METHOD INTERNAL ParseResponsePayload : DINT
VAR_INPUT
  /// Response data
  ResponseData : RobotLibraryRecvDataFB;
  /// Timestamp
  Timestamp    : SystemTime;  
END_VAR
// Table 6-147: Received CMD payload (RC to PLC) of "WriteRobotDefaultDynamics"
// --------------------------
// Header
// --------------------------
// Byte 00 : USINT   - ParSeq | State     
// Byte 01 : SINT    - AlarmMessageSeverity    
// Byte 02 : UINT    - AlarmMessageCode HB
// Byte 03 :         - AlarmMessageCode LB
// --------------------------
// Datablock
// --------------------------
// Byte 04 : UINT VelocityRate
// Byte 05 : 
// Byte 06 : UINT AccelerationRate
// Byte 07 : 
// Byte 08 : UINT DecelerationRate
// Byte 09 : 
// Byte 10 : UINT JerkRate
// Byte 11 : 
// --------------------------
// call base implementation to parse the header from payload buffer
ResponseData.PayloadPtr := SUPER^.ParseResponsePayload(ResponseData := ResponseData, Timestamp := Timestamp);

// copy parsed header to response
_response.ParSeq               := _rspHeader.ParSeq;
_response.State                := _rspHeader.State;
_response.AlarmMessageSeverity := _rspHeader.AlarmMessageSeverity;
_response.AlarmMessageCode     := _rspHeader.AlarmMessageCode;

// Get Response.VelocityRate
_response.VelocityRate     := ResponseData.GetUint();
// Get Response.AccelerationRate
_response.AccelerationRate := ResponseData.GetUint();
// Get Response.DecelerationRate
_response.DecelerationRate := ResponseData.GetUint();
// Get Response.JerkRate
_response.JerkRate         := ResponseData.GetUint();

// Create logging
ParseResponsePayloadLog(ResponseData := ResponseData, Timestamp := Timestamp);
END_METHOD

METHOD INTERNAL ParseResponsePayloadLog
VAR_INPUT
  /// Response data
  ResponseData : RobotLibraryRecvDataFB;
  /// Timestamp
  Timestamp    : SystemTime;  
END_VAR
// Create log entry for Parameter start
CreateLogMessage      ( Timestamp   := Timestamp,
                        MessageType := MessageType.CMD,
                        Severity    := Severity.DEBUG,
                        MessageCode := 0,
                        MessageText := 'Parsed the following parameter(s) from response data:');
               
// Create log entry for VelocityRate
CreateLogMessagePara1 ( Timestamp   := Timestamp,
                        MessageType := MessageType.CMD,
                        Severity    := Severity.DEBUG,
                        MessageCode := 0,
                        MessageText := 'Response.VelocityRate = {1}',
                        Para1       :=  UINT_TO_STRING(_response.VelocityRate));

// Create log entry for AccelerationRate
CreateLogMessagePara1 ( Timestamp   := Timestamp,
                        MessageType := MessageType.CMD,
                        Severity    := Severity.DEBUG,
                        MessageCode := 0,
                        MessageText := 'Response.AccelerationRate = {1}',
                        Para1       :=  UINT_TO_STRING(_response.AccelerationRate));

// Create log entry for DecelerationRate
CreateLogMessagePara1 ( Timestamp   := Timestamp,
                        MessageType := MessageType.CMD,
                        Severity    := Severity.DEBUG,
                        MessageCode := 0,
                        MessageText := 'Response.DecelerationRate = {1}',
                        Para1       :=  UINT_TO_STRING(_response.DecelerationRate));

// Create log entry for JerkRate
CreateLogMessagePara1 ( Timestamp   := Timestamp,
                        MessageType := MessageType.CMD,
                        Severity    := Severity.DEBUG,
                        MessageCode := 0,
                        MessageText := 'Response.JerkRate = {1}',
                        Para1       :=  UINT_TO_STRING(_response.JerkRate));
END_METHOD

METHOD PROTECTED Reset : DINT
VAR_INPUT
END_VAR
Reset := SUPER^.Reset();

Done               := FALSE;
Busy               := FALSE;
CommandBuffered    := FALSE;
CommandAborted     := FALSE;
CommandInterrupted := FALSE;
END_METHOD

END_FUNCTION_BLOCK

// Library/POUs/Write/MC_WriteRobotReferenceDynamics/MC_WriteRobotReferenceDynamicsFB
/// Write reference values of robot dynamics for path movement
FUNCTION_BLOCK MC_WriteRobotReferenceDynamicsFB EXTENDS RobotLibraryBaseExecuteFB
// ------------------------------------------------------------------------- 
//  SRCI Robot Library                                                
// ------------------------------------------------------------------------- 
//                                                                           
//  Object:      WriteRobotReferenceDynamicsFB                                       
//  Author:      Thorsten Brach                                                
//  Date:        2024-06-01
//
//  Description:                                              
//   
//                                                                           
//  Copyright: 
//    (C) 2024 Thorsten Brach. All rights reserved                                                                                                                                            
//             Licensed under the LGPL-3.0 license.
//                                                                           
//  Disclaimer:                                                                           
//    This project is provided without any guarantee and can be used for   
//    private and commercial purposes. Any use is at the user’s 
//    own risk and responsibility.
//
// -------------------------------------------------------------------------
VAR_INPUT
  /// Processing Mode
  ProcessingMode     : ProcessingMode;
  /// internal copy of command parameter 
  ParCmd             : WriteRobotReferenceDynamicsParCmd; 
END_VAR
VAR_OUTPUT
  /// Command is transferred and confirmed by the RC
  CommandBuffered    : BOOL;
  /// The command was aborted by another command
  CommandAborted     : BOOL;
  /// TRUE, while command is interrupted during execution and can be continued.
  CommandInterrupted : BOOL;
  /// command outputs
  OutCmd             : WriteRobotReferenceDynamicsOutCmd;       
END_VAR

VAR
  /// internal copy of command parameter 
 _parCmd             : WriteRobotReferenceDynamicsParCmd;
  /// command data to send
 _command            : WriteRobotReferenceDynamicsSendData;
  /// response data received
 _response           : WriteRobotReferenceDynamicsRecvData;      
END_VAR

SUPER^(AxesGroup := AxesGroup);

METHOD PROTECTED CheckFunctionSupported : BOOL
VAR_IN_OUT
  /// Robot assignment of function
  AxesGroup : AxesGroup; 
END_VAR
CheckFunctionSupported := AxesGroup.InternalData.RCSupportedFunctions.WriteRobotReferenceDynamics;

IF ( NOT CheckFunctionSupported )
THEN
  // call base implementation for set error and create log entry
  SUPER^.CheckFunctionSupported(AxesGroup := AxesGroup);
END_IF
END_METHOD

METHOD PROTECTED CheckParameterChanged : BOOL
VAR_IN_OUT
  /// Robot assignment of function
  AxesGroup    : AxesGroup; 
END_VAR
// Check ParCmd Size is > 0, because MemCmp does not work correctly with size = 0
IF (SIZEOF(ParCmd) = 0) 
THEN 
  RETURN;
END_IF

// compare memory 
_parameterChanged := ( SysDepMemCmp(pData1 := ADR(ParCmd), pData2 := ADR(_parCmd), DataLen := SIZEOF(ParCmd)) <> RobotLibraryConstants.OK );

// check parameter valid ?
_parameterValid   := CheckParameterValid( AxesGroup := AxesGroup );

IF ((  _parameterChanged        )  AND 
    (  _parameterValid          )) OR
    (  _parameterUpdateInternal )  
THEN  
  // reset internal flag for send parameter update
 _parameterUpdateInternal := FALSE;
  // update internal copy of parameters 
 _parCmd := ParCmd;
  // inc parameter sequence
 _command.ParSeq := _command.ParSeq + 1;
  // update command data  
  CommandData := CreateCommandPayload(AxesGroup := AxesGroup); // ( Access via reference to rCommandFB in ACR )
  // notify active command register 
  AxesGroup.Acyclic.ActiveCommandRegister.NotifyParameterChanged := _uniqueID;
END_IF
END_METHOD

METHOD INTERNAL CreateCommandPayload : RobotLibrarySendDataFB
VAR_IN_OUT
  /// Robot assignment of function
  AxesGroup : AxesGroup; 
END_VAR
// Table 6-139: Sent CMD payload (PLC to RC) of "WriteRobotReferenceDynamics"
// --------------------------
// Header
// --------------------------
// Byte 00 : UINT  - Type HB     
// Byte 01 :       - Type LB    
// Byte 02 : USINT - Reserve | ExecutionMode
// Byte 03 : USINT - ParSeq  | Priority
// --------------------------
// Datablock
// --------------------------
// Byte 04 : DATE Date
// Byte 05 : 
// Byte 06 : TIME_OF_DAY Time
// Byte 07 : 
// Byte 08 : 
// Byte 09 : REAL VelocityReference
// Byte 10 : 
// Byte 11 : 
// Byte 12 : REAL AccelerationReference
// Byte 13 : 
// Byte 14 : 
// Byte 15 : REAL DecelerationReference
// Byte 16 : 
// Byte 17 : 
// Byte 18 : REAL JerkReference
// Byte 19 : 
// Byte 20 : 
// Byte 21 : 
// Byte 22 : REAL 
// Byte 23 : 
// Byte 24 : 
// Byte 25 : 
// --------------------------
// set command parameter 
_command.CmdTyp                :=  CmdType.WriteRobotReferenceDynamics;
_command.ExecMode              :=  ExecMode;
_command.ParSeq                := _command.ParSeq;
_command.Priority              :=  Priority;

_command.DynamicValues         := _parCmd.DynamicValues; {warning 'ToDo: Check if this is a mistake in the SRCI specification ? '}

(*
 _command.Timestamp             := _parCmd.DynamicValues.Timestamp;
 _command.VelocityReference     := REAL_TO_PERCENT_UINT(_parCmd.DynamicValues.VelocityReference     , IsOptional := FALSE);
 _command.AccelerationReference := REAL_TO_PERCENT_UINT(_parCmd.DynamicValues.AccelerationReference , IsOptional := FALSE);
 _command.JerkReference         := REAL_TO_PERCENT_UINT(_parCmd.DynamicValues.JerkReference         , IsOptional := TRUE );
 _command.DecelerationReference := REAL_TO_PERCENT_UINT(_parCmd.DynamicValues.DecelerationReference , IsOptional := TRUE );
*)


// copy command data to header
_cmdHeader := _command;
// call base implementation to copy header to payload buffer
CreateCommandPayload := SUPER^.CreateCommandPayload(AxesGroup := AxesGroup);

// add command.DynamicValues.Timestamp.IEC_DATE
CreateCommandPayload.AddUint(_command.DynamicValues.Timestamp.IEC_DATE);
// add command.DynamicValues.Timestamp.IEC_TIME
CreateCommandPayload.AddTime(_command.DynamicValues.Timestamp.IEC_TIME);
// add command.DynamicValues.VelocityReference
CreateCommandPayload.AddReal(_command.DynamicValues.VelocityReference);
// add command.DynamicValues.AccelerationReference
CreateCommandPayload.AddReal(_command.DynamicValues.AccelerationReference);
// add command.DynamicValues.DecelerationRate
CreateCommandPayload.AddReal(_command.DynamicValues.DecelerationReference);
// add command.DynamicValues.JerkRate
CreateCommandPayload.AddReal(_command.DynamicValues.JerkReference);

// Create logging
CreateCommandPayloadLog(AxesGroup := AxesGroup);
END_METHOD

METHOD INTERNAL CreateCommandPayloadLog
VAR_IN_OUT
  /// Robot assignment of function
  AxesGroup : AxesGroup; 
END_VAR
// Create log entry for Parameter start
CreateLogMessage      ( Timestamp   := AxesGroup.InternalData.SystemTime,
                        MessageType := MessageType.CMD,
                        Severity    := Severity.DEBUG,
                        MessageCode := 0,
                        MessageText := 'Create command payload with the following parameter(s) :');
  
// Create log entry for DynamicValues.Timestamp.IEC_DATE
CreateLogMessagePara1 ( Timestamp   := AxesGroup.InternalData.SystemTime,
                        MessageType := MessageType.CMD,
                        Severity    := Severity.DEBUG,
                        MessageCode := 0,
                        MessageText := 'Command.DynamicValues.Timestamp.IEC_DATE = {1}',
                        Para1       :=  IEC_DATE_TO_STRING(_command.DynamicValues.Timestamp.IEC_DATE));

// Create log entry for DynamicValues.Timestamp.IEC_TIME
CreateLogMessagePara1 ( Timestamp   := AxesGroup.InternalData.SystemTime,
                        MessageType := MessageType.CMD,
                        Severity    := Severity.DEBUG,
                        MessageCode := 0,
                        MessageText := 'Command.DynamicValues.Timestamp.IEC_TIME = {1}',
                        Para1       :=  IEC_TIME_TO_STRING(_command.DynamicValues.Timestamp.IEC_TIME));

// Create log entry for DynamicValues.VelocityReference
CreateLogMessagePara1 ( Timestamp   := AxesGroup.InternalData.SystemTime,
                        MessageType := MessageType.CMD,
                        Severity    := Severity.DEBUG,
                        MessageCode := 0,
                        MessageText := 'Command..DynamicValues.VelocityReference = {1}',
                        Para1       :=  REAL_TO_STRING(_command.DynamicValues.VelocityReference));

// Create log entry for DynamicValues.AccelerationReference
CreateLogMessagePara1 ( Timestamp   := AxesGroup.InternalData.SystemTime,
                        MessageType := MessageType.CMD,
                        Severity    := Severity.DEBUG,
                        MessageCode := 0,
                        MessageText := 'Command.DynamicValues.AccelerationReference = {1}',
                        Para1       :=  REAL_TO_STRING(_command.DynamicValues.AccelerationReference));

// Create log entry for DynamicValues.DecelerationReference
CreateLogMessagePara1 ( Timestamp   := AxesGroup.InternalData.SystemTime,
                        MessageType := MessageType.CMD,
                        Severity    := Severity.DEBUG,
                        MessageCode := 0,
                        MessageText := 'Command.DynamicValues.DecelerationReference = {1}',
                        Para1       :=  REAL_TO_STRING(_command.DynamicValues.DecelerationReference));

// Create log entry for DynamicValues.JerkReference
CreateLogMessagePara1 ( Timestamp   := AxesGroup.InternalData.SystemTime,
                        MessageType := MessageType.CMD,
                        Severity    := Severity.DEBUG,
                        MessageCode := 0,
                        MessageText := 'Command.DynamicValues.JerkReference = {1}',
                        Para1       :=  REAL_TO_STRING(_command.DynamicValues.JerkReference));
END_METHOD

METHOD FB_init : BOOL
VAR_INPUT
  /// if TRUE, the retain variables are initialized (warm start / cold start)
  bInitRetains : BOOL; 
  /// if TRUE, the instance afterwards gets moved into the copy code (online change)
  bInCopyCode  : BOOL;  
END_VAR
MyType := 'MC_WriteRobotReferenceDynamicsFB';

ExecMode := ExecutionMode.PARALLEL;
END_METHOD

METHOD PROTECTED OnCall
VAR_IN_OUT
  /// Robot assignment of function
  AxesGroup : AxesGroup; 
END_VAR
// call base implementation
SUPER^.OnCall(AxesGroup := AxesGroup);

CASE _stepCmd OF
  
  00:  IF ( _execute_R.Q )  
       THEN
         // Check function is supported and parameter are valid ?
         IF (( CheckFunctionSupported( AxesGroup := AxesGroup )) AND
             ( CheckParameterValid   ( AxesGroup := AxesGroup )))
         THEN      
           // set busy flag
           Busy := TRUE;
           // Reset command outputs
           SysDepMemSet(pDest := ADR(OutCmd), Value := 0, DataLen := SIZEOF(OutCmd));         
           // apply command parameter
          _parCmd := ParCmd;
           // init parameter sequence
          _command.ParSeq := 1;
           // create command data
           CommandData := CreateCommandPayload(AxesGroup := AxesGroup);
           // Add command to active command register
          _uniqueID := AxesGroup.Acyclic.ActiveCommandRegister.AddCmd( pCommandFB := ADR(THIS^ ));     
           // set timeout
           SetTimeout(PT := _timeoutCmd, rTimer := _timerCmd);
           // inc step counter
          _stepCmd := _stepCmd + 1;
         END_IF 
       END_IF
     

  01:  // Wait for responce received
       IF ( _responseReceived )
       THEN
         // reset response received flag
        _responseReceived := FALSE;

         CASE  _response.State 
         OF
           CmdMessageState.BUFFERED    : CommandBuffered    := TRUE;
           CmdMessageState.INTERRUPTED : CommandInterrupted := TRUE;           
           CmdMessageState.DONE        : Done               := TRUE;           
           CmdMessageState.ABORTED     : CommandAborted     := TRUE;
           CmdMessageState.ERROR       : Error              := TRUE;
         END_CASE
                
         // Done, Aborted or Error ?
         IF (_response.State >= CmdMessageState.DONE )
         THEN
           // Reset Busy flag
           Busy := FALSE;
           // Update results
           OutCmd.ReferenceDynamicValues.VelocityReference     := _response.ReferenceDynamicValues.VelocityReference; 
           OutCmd.ReferenceDynamicValues.AccelerationReference := _response.ReferenceDynamicValues.AccelerationReference;
           OutCmd.ReferenceDynamicValues.DecelerationReference := _response.ReferenceDynamicValues.DecelerationReference;
           OutCmd.ReferenceDynamicValues.JerkReference         := _response.ReferenceDynamicValues.JerkReference;

           // set timeout
           SetTimeout(PT := _timeoutCmd, rTimer := _timerCmd);
           // inc step counter
          _stepCmd := _stepCmd + 1; 
         END_IF
       END_IF


  02: IF ( NOT Execute)
      THEN
        Reset();
      END_IF     

ELSE
  // invalid step
  ErrorID := RobotLibraryEvents.ERR_INVALID_STEP;
END_CASE


// Reset FB
IF ( NOT Execute )
THEN
  Reset();
END_IF
END_METHOD

METHOD INTERNAL ParseResponsePayload : DINT
VAR_INPUT
  /// Response data
  ResponseData : RobotLibraryRecvDataFB;
  /// Timestamp
  Timestamp    : SystemTime;  
END_VAR
// Table 6-140: Received CMD payload (RC to PLC) of "WriteRobotReferenceDynamics"
// --------------------------
// Header
// --------------------------
// Byte 00 : USINT   - ParSeq | State     
// Byte 01 : SINT    - AlarmMessageSeverity    
// Byte 02 : UINT    - AlarmMessageCode HB
// Byte 03 :         - AlarmMessageCode LB
// --------------------------
// Datablock
// --------------------------
// Byte 04 : REAL VelocityReference
// Byte 05 : 
// Byte 06 : 
// Byte 07 : 
// Byte 08 : REAL AccelerationReference
// Byte 09 : 
// Byte 10 : 
// Byte 11 : 
// Byte 12 : REAL DecelerationReference
// Byte 13 : 
// Byte 14 : 
// Byte 15 : 
// Byte 16 : REAL JerkReference
// Byte 17 : 
// Byte 18 : 
// Byte 19 : 
// --------------------------
// call base implementation to parse the header from payload buffer
ResponseData.PayloadPtr := SUPER^.ParseResponsePayload(ResponseData := ResponseData, Timestamp := Timestamp);

// copy parsed header to response
_response.ParSeq               := _rspHeader.ParSeq;
_response.State                := _rspHeader.State;
_response.AlarmMessageSeverity := _rspHeader.AlarmMessageSeverity;
_response.AlarmMessageCode     := _rspHeader.AlarmMessageCode;

// Get Response.ReferenceDynamicValues.VelocityReference
_response.ReferenceDynamicValues.VelocityReference := ResponseData.GetReal();
// Get Response.ReferenceDynamicValues.AccelerationReference
_response.ReferenceDynamicValues.AccelerationReference := ResponseData.GetReal();
// Get Response.ReferenceDynamicValues.DecelerationReference
_response.ReferenceDynamicValues.DecelerationReference := ResponseData.GetReal();
// Get ReferenceDynamicValues.JerkReference
_response.ReferenceDynamicValues.JerkReference := ResponseData.GetReal();

// Create logging
ParseResponsePayloadLog(ResponseData := ResponseData, Timestamp := Timestamp);
END_METHOD

METHOD INTERNAL ParseResponsePayloadLog
VAR_INPUT
  /// Response data
  ResponseData : RobotLibraryRecvDataFB;
  /// Timestamp
  Timestamp    : SystemTime;  
END_VAR
// Create log entry for Parameter start
CreateLogMessage      ( Timestamp   := Timestamp,
                        MessageType := MessageType.CMD,
                        Severity    := Severity.DEBUG,
                        MessageCode := 0,
                        MessageText := 'Parsed the following parameter(s) from response data:');

// Create log entry for ReferenceDynamicValues.VelocityReference
CreateLogMessagePara1 ( Timestamp   := Timestamp,
                        MessageType := MessageType.CMD,
                        Severity    := Severity.DEBUG,
                        MessageCode := 0,
                        MessageText := 'Response.ReferenceDynamicValues.VelocityReference = {1}',
                        Para1       :=  REAL_TO_STRING(_response.ReferenceDynamicValues.VelocityReference));

// Create log entry for ReferenceDynamicValues.AccelerationReference
CreateLogMessagePara1 ( Timestamp   := Timestamp,
                        MessageType := MessageType.CMD,
                        Severity    := Severity.DEBUG,
                        MessageCode := 0,
                        MessageText := 'Response.ReferenceDynamicValues.AccelerationReference = {1}',
                        Para1       :=  REAL_TO_STRING(_response.ReferenceDynamicValues.AccelerationReference));
                        
// Create log entry for ReferenceDynamicValues.DecelerationReference
CreateLogMessagePara1 ( Timestamp   := Timestamp,
                        MessageType := MessageType.CMD,
                        Severity    := Severity.DEBUG,
                        MessageCode := 0,
                        MessageText := 'Response.ReferenceDynamicValues.DecelerationReference = {1}',
                        Para1       :=  REAL_TO_STRING(_response.ReferenceDynamicValues.DecelerationReference));

// Create log entry for ReferenceDynamicValues.JerkReference
CreateLogMessagePara1 ( Timestamp   := Timestamp,
                        MessageType := MessageType.CMD,
                        Severity    := Severity.DEBUG,
                        MessageCode := 0,
                        MessageText := 'Response.ReferenceDynamicValues.JerkReference = {1}',
                        Para1       :=  REAL_TO_STRING(_response.ReferenceDynamicValues.JerkReference));
END_METHOD

METHOD PROTECTED Reset : DINT
VAR_INPUT
END_VAR
Reset := SUPER^.Reset();

Done               := FALSE;
Busy               := FALSE;
CommandBuffered    := FALSE;
CommandAborted     := FALSE;
CommandInterrupted := FALSE;
END_METHOD

END_FUNCTION_BLOCK

// Library/POUs/Write/MC_WriteRobotSWLimits/MC_WriteRobotSWLimitsFB
/// Change robot limits of robot axes (degree)
FUNCTION_BLOCK MC_WriteRobotSWLimitsFB EXTENDS RobotLibraryBaseExecuteFB
// ------------------------------------------------------------------------- 
//  SRCI Robot Library                                                
// ------------------------------------------------------------------------- 
//                                                                           
//  Object:      WriteRobotSWLimitsFB                                       
//  Author:      Thorsten Brach                                                
//  Date:        2024-06-01
//
//  Description:                                              
//   
//                                                                           
//  Copyright: 
//    (C) 2024 Thorsten Brach. All rights reserved                                                                                                                                            
//             Licensed under the LGPL-3.0 license.
//                                                                           
//  Disclaimer:                                                                           
//    This project is provided without any guarantee and can be used for   
//    private and commercial purposes. Any use is at the user’s 
//    own risk and responsibility.
//
// -------------------------------------------------------------------------
VAR_INPUT
  /// command parameter 
  ParCmd          : WriteRobotSWLimitsParCmd;
END_VAR
VAR_OUTPUT
  /// Command is transferred and confirmed by the RC
  CommandBuffered : BOOL;
  /// command outputs
  OutCmd          : WriteRobotSWLimitsOutCmd;       
END_VAR

VAR
  /// internal copy of command parameter 
 _parCmd          : WriteRobotSWLimitsParCmd;
  /// command data to send
 _command         : WriteRobotSWLimitsSendData;
  /// response data received
 _response        : WriteRobotSWLimitsRecvData;      
END_VAR

SUPER^(AxesGroup := AxesGroup);

METHOD PROTECTED CheckFunctionSupported : BOOL
VAR_IN_OUT
  /// Robot assignment of function
  AxesGroup : AxesGroup; 
END_VAR
CheckFunctionSupported := AxesGroup.InternalData.RCSupportedFunctions.WriteRobotSWLimits;

IF ( NOT CheckFunctionSupported )
THEN
  // call base implementation for set error and create log entry
  SUPER^.CheckFunctionSupported(AxesGroup := AxesGroup);
END_IF
END_METHOD

METHOD PROTECTED CheckParameterChanged : BOOL
VAR_IN_OUT
  /// Robot assignment of function
  AxesGroup    : AxesGroup; 
END_VAR
// Check ParCmd Size is > 0, because MemCmp does not work correctly with size = 0
IF (SIZEOF(ParCmd) = 0) 
THEN 
  RETURN;
END_IF

// compare memory 
_parameterChanged := ( SysDepMemCmp(pData1 := ADR(ParCmd), pData2 := ADR(_parCmd), DataLen := SIZEOF(ParCmd)) <> RobotLibraryConstants.OK );

// check parameter valid ?
_parameterValid   := CheckParameterValid( AxesGroup := AxesGroup );

IF ((  _parameterChanged        )  AND 
    (  _parameterValid          )) OR
    (  _parameterUpdateInternal )  
THEN  
  // reset internal flag for send parameter update
 _parameterUpdateInternal := FALSE;
  // update internal copy of parameters 
 _parCmd := ParCmd;
  // inc parameter sequence
 _command.ParSeq := _command.ParSeq + 1;
  // update command data  
  CommandData := CreateCommandPayload(AxesGroup := AxesGroup); // ( Access via reference to rCommandFB in ACR )
  // notify active command register 
  AxesGroup.Acyclic.ActiveCommandRegister.NotifyParameterChanged := _uniqueID;
END_IF
END_METHOD

METHOD INTERNAL CreateCommandPayload : RobotLibrarySendDataFB
VAR_IN_OUT
  /// Robot assignment of function
  AxesGroup : AxesGroup; 
END_VAR
// Table 6-185: Sent CMD payload (PLC to RC) of "WriteRobotSWLimits"
// --------------------------
// Header
// --------------------------
// Byte 00 : UINT  - Type HB     
// Byte 01 :       - Type LB    
// Byte 02 : USINT - Reserve | ExecutionMode
// Byte 03 : USINT - ParSeq  | Priority
// --------------------------
// Datablock
// --------------------------
// Byte 04 : DATE Date
// Byte 05 : 
// Byte 06 : TIME_OF_DAY Time
// Byte 07 : 
// Byte 08 : 
// Byte 09 : REAL J1LowerLimit
// Byte 10 : 
// Byte 11 : 
// Byte 12 : REAL J2LowerLimit
// Byte 13 : 
// Byte 14 : 
// Byte 15 : REAL J3LowerLimit
// Byte 16 : 
// Byte 17 : 
// Byte 18 : REAL J4LowerLimit
// Byte 19 : 
// Byte 20 : 
// Byte 21 : REAL J5LowerLimit
// Byte 22 : 
// Byte 23 : 
// Byte 24 : REAL J6LowerLimit
// Byte 25 : 
// Byte 26 : 
// Byte 27 : REAL E1LowerLimit
// Byte 28 : 
// Byte 29 : 
// Byte 30 : REAL J1UpperLimit
// Byte 31 : 
// Byte 32 : 
// Byte 33 : REAL J2UpperLimit
// Byte 34 : 
// Byte 35 : 
// Byte 36 : REAL J3UpperLimit
// Byte 37 : 
// Byte 38 : 
// Byte 39 : REAL J4UpperLimit
// Byte 40 : 
// Byte 41 : 
// Byte 42 : REAL J5UpperLimit
// Byte 43 : 
// Byte 44 : 
// Byte 45 : REAL J6UpperLimit
// Byte 46 : 
// Byte 47 : 
// Byte 48 : REAL E1UpperLimit
// Byte 49 : 
// Byte 50 : 
// Byte 51 : REAL E2LowerLimit
// Byte 52 : 
// Byte 53 : 
// Byte 54 : REAL E3LowerLimit
// Byte 55 : 
// Byte 56 : 
// Byte 57 : REAL E4LowerLimit
// Byte 58 : 
// Byte 59 : 
// Byte 60 : REAL E5LowerLimit
// Byte 61 : 
// Byte 62 : 
// Byte 63 : REAL E6LowerLimit
// Byte 64 : 
// Byte 65 : 
// Byte 66 : REAL E2UpperLimit
// Byte 67 : 
// Byte 68 : 
// Byte 69 : REAL E3UpperLimit
// Byte 70 : 
// Byte 71 : 
// Byte 72 : REAL E4UpperLimit
// Byte 73 : 
// Byte 74 : 
// Byte 75 : REAL E5UpperLimit
// Byte 76 : 
// Byte 77 : 
// Byte 78 : REAL E6UpperLimit
// Byte 79 : 
// Byte 80 : 
// Byte 81 : 
// Byte 82 : BOOL ResetToFactoryDefault
// --------------------------
// set command parameter 
_command.CmdTyp                 :=  CmdType.WriteRobotSWLimits;
_command.ExecMode               :=  ExecMode;
_command.ParSeq                 := _command.ParSeq;
_command.Priority               :=  Priority;
                                
_command.LimitValues            :=  _parCmd.LimitValues;
_command.ResetToFactoryDefaults :=  _parCmd.ResetToFactoryDefaults;

// copy command data to header
_cmdHeader := _command;
// call base implementation to copy header to payload buffer
CreateCommandPayload := SUPER^.CreateCommandPayload(AxesGroup := AxesGroup);

// add command.LimitValues.Timestamp.IEC_DATE
CreateCommandPayload.AddUint(_command.LimitValues.Timestamp.IEC_DATE);
// add command.LimitValues.Timestamp.IEC_TIME
CreateCommandPayload.AddTime(_command.LimitValues.Timestamp.IEC_TIME);
// add command.LimitValues.J1LowerLimit
CreateCommandPayload.AddReal(_command.LimitValues.J1LowerLimit);
// add command.LimitValues.J2LowerLimit
CreateCommandPayload.AddReal(_command.LimitValues.J2LowerLimit);
// add command.LimitValues.J3LowerLimit
CreateCommandPayload.AddReal(_command.LimitValues.J3LowerLimit);
// add command.LimitValues.J41LowerLimit
CreateCommandPayload.AddReal(_command.LimitValues.J4LowerLimit);
// add command.LimitValues.J5LowerLimit
CreateCommandPayload.AddReal(_command.LimitValues.J5LowerLimit);
// add command.LimitValues.J6LowerLimit
CreateCommandPayload.AddReal(_command.LimitValues.J6LowerLimit);
// add command.LimitValues.E1LowerLimit
CreateCommandPayload.AddReal(_command.LimitValues.E1LowerLimit);
// add command.LimitValues.J1UpperLimit
CreateCommandPayload.AddReal(_command.LimitValues.J1UpperLimit);
// add command.LimitValues.J2UpperLimit
CreateCommandPayload.AddReal(_command.LimitValues.J2UpperLimit);
// add command.LimitValues.J3UpperLimit
CreateCommandPayload.AddReal(_command.LimitValues.J3UpperLimit);
// add command.LimitValues.J4UpperLimit
CreateCommandPayload.AddReal(_command.LimitValues.J4UpperLimit);
// add command.LimitValues.J5UpperLimit
CreateCommandPayload.AddReal(_command.LimitValues.J5UpperLimit);
// add command.LimitValues.J6UpperLimit
CreateCommandPayload.AddReal(_command.LimitValues.J6UpperLimit);
// add command.LimitValues.E1UpperLimit
CreateCommandPayload.AddReal(_command.LimitValues.E1UpperLimit);
// add command.LimitValues.E2LowerLimit
CreateCommandPayload.AddReal(_command.LimitValues.E2LowerLimit);
// add command.LimitValues.E3LowerLimit
CreateCommandPayload.AddReal(_command.LimitValues.E3LowerLimit);
// add command.LimitValues.E4LowerLimit
CreateCommandPayload.AddReal(_command.LimitValues.E4LowerLimit);
// add command.LimitValues.E5LowerLimit
CreateCommandPayload.AddReal(_command.LimitValues.E5LowerLimit);
// add command.LimitValues.E6LowerLimit
CreateCommandPayload.AddReal(_command.LimitValues.E6LowerLimit);
// add command.LimitValues.E2UpperLimit
CreateCommandPayload.AddReal(_command.LimitValues.E2UpperLimit);
// add command.LimitValues.E3UpperLimit
CreateCommandPayload.AddReal(_command.LimitValues.E3UpperLimit);
// add command.LimitValues.E4UpperLimit
CreateCommandPayload.AddReal(_command.LimitValues.E4UpperLimit);
// add command.LimitValues.E5UpperLimit
CreateCommandPayload.AddReal(_command.LimitValues.E5UpperLimit);
// add command.LimitValues.E6UpperLimit
CreateCommandPayload.AddReal(_command.LimitValues.E6UpperLimit);

// Create logging
CreateCommandPayloadLog(AxesGroup := AxesGroup);
END_METHOD

METHOD INTERNAL CreateCommandPayloadLog
VAR_IN_OUT
  /// Robot assignment of function
  AxesGroup : AxesGroup; 
END_VAR
// Create log entry for Parameter start
CreateLogMessage      ( Timestamp   := AxesGroup.InternalData.SystemTime,
                        MessageType := MessageType.CMD,
                        Severity    := Severity.DEBUG,
                        MessageCode := 0,
                        MessageText := 'Create command payload with the following parameter(s) :');
  
// Create log entry for LimitValues.Timestamp.IEC_DATE
CreateLogMessagePara1 ( Timestamp   := AxesGroup.InternalData.SystemTime,
                        MessageType := MessageType.CMD,
                        Severity    := Severity.DEBUG,
                        MessageCode := 0,
                        MessageText := 'Command.LimitValues.Timestamp.IEC_DATE = {1}',
                        Para1       :=  IEC_DATE_TO_STRING(_command.LimitValues.Timestamp.IEC_DATE));

// Create log entry for LimitValues.Timestamp.IEC_TIME
CreateLogMessagePara1 ( Timestamp   := AxesGroup.InternalData.SystemTime,
                        MessageType := MessageType.CMD,
                        Severity    := Severity.DEBUG,
                        MessageCode := 0,
                        MessageText := 'Command.LimitValues.Timestamp.IEC_TIME = {1}',
                        Para1       :=  IEC_TIME_TO_STRING(_command.LimitValues.Timestamp.IEC_TIME));

// Create log entry for LimitValues.J1LowerLimit
CreateLogMessagePara1 ( Timestamp   := AxesGroup.InternalData.SystemTime,
                        MessageType := MessageType.CMD,
                        Severity    := Severity.DEBUG,
                        MessageCode := 0,
                        MessageText := 'Command.LimitValues.J1LowerLimit = {1}',
                        Para1       :=  REAL_TO_STRING(_command.LimitValues.J1LowerLimit));

// Create log entry for LimitValues.J2LowerLimit
CreateLogMessagePara1 ( Timestamp   := AxesGroup.InternalData.SystemTime,
                        MessageType := MessageType.CMD,
                        Severity    := Severity.DEBUG,
                        MessageCode := 0,
                        MessageText := 'Command.LimitValues.J2LowerLimit = {1}',
                        Para1       :=  REAL_TO_STRING(_command.LimitValues.J2LowerLimit));
                        
// Create log entry for LimitValues.J3LowerLimit
CreateLogMessagePara1 ( Timestamp   := AxesGroup.InternalData.SystemTime,
                        MessageType := MessageType.CMD,
                        Severity    := Severity.DEBUG,
                        MessageCode := 0,
                        MessageText := 'Command.LimitValues.J3LowerLimit = {1}',
                        Para1       :=  REAL_TO_STRING(_command.LimitValues.J3LowerLimit));
                        
// Create log entry for LimitValues.J4LowerLimit
CreateLogMessagePara1 ( Timestamp   := AxesGroup.InternalData.SystemTime,
                        MessageType := MessageType.CMD,
                        Severity    := Severity.DEBUG,
                        MessageCode := 0,
                        MessageText := 'Command.LimitValues.J4LowerLimit = {1}',
                        Para1       :=  REAL_TO_STRING(_command.LimitValues.J4LowerLimit));

// Create log entry for LimitValues.J5LowerLimit
CreateLogMessagePara1 ( Timestamp   := AxesGroup.InternalData.SystemTime,
                        MessageType := MessageType.CMD,
                        Severity    := Severity.DEBUG,
                        MessageCode := 0,
                        MessageText := 'Command.LimitValues.J5LowerLimit = {1}',
                        Para1       :=  REAL_TO_STRING(_command.LimitValues.J5LowerLimit));

// Create log entry for LimitValues.J6LowerLimit
CreateLogMessagePara1 ( Timestamp   := AxesGroup.InternalData.SystemTime,
                        MessageType := MessageType.CMD,
                        Severity    := Severity.DEBUG,
                        MessageCode := 0,
                        MessageText := 'Command.LimitValues.J6LowerLimit = {1}',
                        Para1       :=  REAL_TO_STRING(_command.LimitValues.J6LowerLimit));

// Create log entry for LimitValues.E1LowerLimit
CreateLogMessagePara1 ( Timestamp   := AxesGroup.InternalData.SystemTime,
                        MessageType := MessageType.CMD,
                        Severity    := Severity.DEBUG,
                        MessageCode := 0,
                        MessageText := 'Command.LimitValues.E1LowerLimit = {1}',
                        Para1       :=  REAL_TO_STRING(_command.LimitValues.E1LowerLimit));

// Create log entry for LimitValues.J1UpperLimit
CreateLogMessagePara1 ( Timestamp   := AxesGroup.InternalData.SystemTime,
                        MessageType := MessageType.CMD,
                        Severity    := Severity.DEBUG,
                        MessageCode := 0,
                        MessageText := 'Command.LimitValues.J1UpperLimit = {1}',
                        Para1       :=  REAL_TO_STRING(_command.LimitValues.J1UpperLimit));

// Create log entry for LimitValues.J2UpperLimit
CreateLogMessagePara1 ( Timestamp   := AxesGroup.InternalData.SystemTime,
                        MessageType := MessageType.CMD,
                        Severity    := Severity.DEBUG,
                        MessageCode := 0,
                        MessageText := 'Command.LimitValues.J2UpperLimit = {1}',
                        Para1       :=  REAL_TO_STRING(_command.LimitValues.J2UpperLimit));

// Create log entry for LimitValues.J3UpperLimit
CreateLogMessagePara1 ( Timestamp   := AxesGroup.InternalData.SystemTime,
                        MessageType := MessageType.CMD,
                        Severity    := Severity.DEBUG,
                        MessageCode := 0,
                        MessageText := 'Command.LimitValues.J3UpperLimit = {1}',
                        Para1       :=  REAL_TO_STRING(_command.LimitValues.J3UpperLimit));

// Create log entry for LimitValues.J4UpperLimit
CreateLogMessagePara1 ( Timestamp   := AxesGroup.InternalData.SystemTime,
                        MessageType := MessageType.CMD,
                        Severity    := Severity.DEBUG,
                        MessageCode := 0,
                        MessageText := 'Command.LimitValues.J4UpperLimit = {1}',
                        Para1       :=  REAL_TO_STRING(_command.LimitValues.J4UpperLimit));

// Create log entry for LimitValues.J5UpperLimit
CreateLogMessagePara1 ( Timestamp   := AxesGroup.InternalData.SystemTime,
                        MessageType := MessageType.CMD,
                        Severity    := Severity.DEBUG,
                        MessageCode := 0,
                        MessageText := 'Command.LimitValues.J5UpperLimit = {1}',
                        Para1       :=  REAL_TO_STRING(_command.LimitValues.J5UpperLimit));

// Create log entry for LimitValues.J6UpperLimit
CreateLogMessagePara1 ( Timestamp   := AxesGroup.InternalData.SystemTime,
                        MessageType := MessageType.CMD,
                        Severity    := Severity.DEBUG,
                        MessageCode := 0,
                        MessageText := 'Command.LimitValues.J6UpperLimit = {1}',
                        Para1       :=  REAL_TO_STRING(_command.LimitValues.J6UpperLimit));

// Create log entry for LimitValues.E1UpperLimit
CreateLogMessagePara1 ( Timestamp   := AxesGroup.InternalData.SystemTime,
                        MessageType := MessageType.CMD,
                        Severity    := Severity.DEBUG,
                        MessageCode := 0,
                        MessageText := 'Command.LimitValues.E1UpperLimit = {1}',
                        Para1       :=  REAL_TO_STRING(_command.LimitValues.E1UpperLimit));

// Create log entry for LimitValues.E2LowerLimit
CreateLogMessagePara1 ( Timestamp   := AxesGroup.InternalData.SystemTime,
                        MessageType := MessageType.CMD,
                        Severity    := Severity.DEBUG,
                        MessageCode := 0,
                        MessageText := 'Command.LimitValues.E2LowerLimit = {1}',
                        Para1       :=  REAL_TO_STRING(_command.LimitValues.E2LowerLimit));

// Create log entry for LimitValues.E3LowerLimit
CreateLogMessagePara1 ( Timestamp   := AxesGroup.InternalData.SystemTime,
                        MessageType := MessageType.CMD,
                        Severity    := Severity.DEBUG,
                        MessageCode := 0,
                        MessageText := 'Command.LimitValues.E3LowerLimit = {1}',
                        Para1       :=  REAL_TO_STRING(_command.LimitValues.E3LowerLimit));

// Create log entry for LimitValues.E4LowerLimit
CreateLogMessagePara1 ( Timestamp   := AxesGroup.InternalData.SystemTime,
                        MessageType := MessageType.CMD,
                        Severity    := Severity.DEBUG,
                        MessageCode := 0,
                        MessageText := 'Command.LimitValues.E4LowerLimit = {1}',
                        Para1       :=  REAL_TO_STRING(_command.LimitValues.E4LowerLimit));

// Create log entry for LimitValues.E5LowerLimit
CreateLogMessagePara1 ( Timestamp   := AxesGroup.InternalData.SystemTime,
                        MessageType := MessageType.CMD,
                        Severity    := Severity.DEBUG,
                        MessageCode := 0,
                        MessageText := 'Command.LimitValues.E5LowerLimit = {1}',
                        Para1       :=  REAL_TO_STRING(_command.LimitValues.E5LowerLimit));

// Create log entry for LimitValues.E6LowerLimit
CreateLogMessagePara1 ( Timestamp   := AxesGroup.InternalData.SystemTime,
                        MessageType := MessageType.CMD,
                        Severity    := Severity.DEBUG,
                        MessageCode := 0,
                        MessageText := 'Command.LimitValues.E6LowerLimit = {1}',
                        Para1       :=  REAL_TO_STRING(_command.LimitValues.E6LowerLimit));

// Create log entry for LimitValues.E2UpperLimit
CreateLogMessagePara1 ( Timestamp   := AxesGroup.InternalData.SystemTime,
                        MessageType := MessageType.CMD,
                        Severity    := Severity.DEBUG,
                        MessageCode := 0,
                        MessageText := 'Command.LimitValues.E2UpperLimit = {1}',
                        Para1       :=  REAL_TO_STRING(_command.LimitValues.E2UpperLimit));

// Create log entry for LimitValues.E3UpperLimit
CreateLogMessagePara1 ( Timestamp   := AxesGroup.InternalData.SystemTime,
                        MessageType := MessageType.CMD,
                        Severity    := Severity.DEBUG,
                        MessageCode := 0,
                        MessageText := 'Command.LimitValues.E3UpperLimit = {1}',
                        Para1       :=  REAL_TO_STRING(_command.LimitValues.E3UpperLimit));                        
                        
// Create log entry for LimitValues.E4UpperLimit
CreateLogMessagePara1 ( Timestamp   := AxesGroup.InternalData.SystemTime,
                        MessageType := MessageType.CMD,
                        Severity    := Severity.DEBUG,
                        MessageCode := 0,
                        MessageText := 'Command.LimitValues.E4UpperLimit = {1}',
                        Para1       :=  REAL_TO_STRING(_command.LimitValues.E4UpperLimit));                                                
                        
// Create log entry for LimitValues.E5UpperLimit
CreateLogMessagePara1 ( Timestamp   := AxesGroup.InternalData.SystemTime,
                        MessageType := MessageType.CMD,
                        Severity    := Severity.DEBUG,
                        MessageCode := 0,
                        MessageText := 'Command.LimitValues.E5UpperLimit = {1}',
                        Para1       :=  REAL_TO_STRING(_command.LimitValues.E5UpperLimit));                                                                        
                        
// Create log entry for LimitValues.E6UpperLimit
CreateLogMessagePara1 ( Timestamp   := AxesGroup.InternalData.SystemTime,
                        MessageType := MessageType.CMD,
                        Severity    := Severity.DEBUG,
                        MessageCode := 0,
                        MessageText := 'Command.LimitValues.E6UpperLimit = {1}',
                        Para1       :=  REAL_TO_STRING(_command.LimitValues.E6UpperLimit));
END_METHOD

METHOD FB_init : BOOL
VAR_INPUT
  /// if TRUE, the retain variables are initialized (warm start / cold start)
  bInitRetains : BOOL; 
  /// if TRUE, the instance afterwards gets moved into the copy code (online change)
  bInCopyCode  : BOOL;  
END_VAR
MyType := 'MC_WriteRobotSWLimitsFB';

ExecMode := ExecutionMode.PARALLEL;
END_METHOD

METHOD PROTECTED OnCall
VAR_IN_OUT
  /// Robot assignment of function
  AxesGroup : AxesGroup; 
END_VAR
// call base implementation
SUPER^.OnCall(AxesGroup := AxesGroup);

CASE _stepCmd OF
  
  00:  IF ( _execute_R.Q )  
       THEN
         // Check function is supported and parameter are valid ?
         IF (( CheckFunctionSupported( AxesGroup := AxesGroup )) AND
             ( CheckParameterValid   ( AxesGroup := AxesGroup )))
         THEN      
           // set busy flag
           Busy := TRUE;
           // Reset command outputs
           SysDepMemSet(pDest := ADR(OutCmd), Value := 0, DataLen := SIZEOF(OutCmd));         
           // apply command parameter
          _parCmd := ParCmd;
           // init parameter sequence
          _command.ParSeq := 1;
           // create command data
           CommandData := CreateCommandPayload(AxesGroup := AxesGroup);
           // Add command to active command register
          _uniqueID := AxesGroup.Acyclic.ActiveCommandRegister.AddCmd( pCommandFB := ADR(THIS^ ));     
           // set timeout
           SetTimeout(PT := _timeoutCmd, rTimer := _timerCmd);
           // inc step counter
          _stepCmd := _stepCmd + 1;
         END_IF 
       END_IF
     

  01:  // Wait for responce received
       IF ( _responseReceived )
       THEN
         // reset response received flag
        _responseReceived := FALSE;

         CASE  _response.State 
         OF
           CmdMessageState.BUFFERED : CommandBuffered := TRUE;
           CmdMessageState.DONE     : Done            := TRUE;
           CmdMessageState.ERROR    : Error           := TRUE;
         END_CASE
                
         // Done, Aborted or Error ?
         IF (_response.State >= CmdMessageState.DONE )
         THEN
           // Reset Busy flag
           Busy := FALSE;
           // Update results
           OutCmd.RestartRequested  := _response.RestartRequested;
           // set timeout
           SetTimeout(PT := _timeoutCmd, rTimer := _timerCmd);
           // inc step counter
          _stepCmd := _stepCmd + 1; 
         END_IF
       END_IF


  02: IF ( NOT Execute)
      THEN
        Reset(); 
      END_IF     

ELSE
  // invalid step
  ErrorID := RobotLibraryEvents.ERR_INVALID_STEP;
END_CASE


// Reset FB
IF ( NOT Execute )
THEN
  Reset(); 
END_IF
END_METHOD

METHOD INTERNAL ParseResponsePayload : DINT
VAR_INPUT
  /// Response data
  ResponseData : RobotLibraryRecvDataFB;
  /// Timestamp
  Timestamp    : SystemTime;  
END_VAR
// Table 6-186: Received CMD payload (RC to PLC) of "WriteRobotSWLimits"
// --------------------------
// Header
// --------------------------
// Byte 00 : USINT   - ParSeq | State     
// Byte 01 : SINT    - AlarmMessageSeverity    
// Byte 02 : UINT    - AlarmMessageCode HB
// Byte 03 :         - AlarmMessageCode LB
// --------------------------
// Datablock
// --------------------------
// Byte 04 : BOOL       - RestartRequested
// call base implementation to parse the header from payload buffer
ResponseData.PayloadPtr := SUPER^.ParseResponsePayload(ResponseData := ResponseData, Timestamp := Timestamp);

// copy parsed header to response
_response.ParSeq               := _rspHeader.ParSeq;
_response.State                := _rspHeader.State;
_response.AlarmMessageSeverity := _rspHeader.AlarmMessageSeverity;
_response.AlarmMessageCode     := _rspHeader.AlarmMessageCode;

// Get Response.RestartRequested
_response.RestartRequested := ResponseData.GetBool();

// Create logging
ParseResponsePayloadLog(ResponseData := ResponseData, Timestamp := Timestamp);
END_METHOD

METHOD INTERNAL ParseResponsePayloadLog
VAR_INPUT
  /// Response data
  ResponseData : RobotLibraryRecvDataFB;
  /// Timestamp
  Timestamp    : SystemTime;  
END_VAR
// Create log entry for Parameter start
CreateLogMessage      ( Timestamp   := Timestamp,
                        MessageType := MessageType.CMD,
                        Severity    := Severity.DEBUG,
                        MessageCode := 0,
                        MessageText := 'Parsed the following parameter(s) from response data:');
        

// Create log entry for RestartRequested
CreateLogMessagePara1 ( Timestamp   := Timestamp,
                        MessageType := MessageType.CMD,
                        Severity    := Severity.DEBUG,
                        MessageCode := 0,
                        MessageText := 'Response.RestartRequested = {1}',
                        Para1       :=  BOOL_TO_STRING(_response.RestartRequested));
END_METHOD

METHOD PROTECTED Reset : DINT
VAR_INPUT
END_VAR
Reset := SUPER^.Reset();

Done               := FALSE;
Busy               := FALSE;
CommandBuffered    := FALSE;
END_METHOD

END_FUNCTION_BLOCK

// Library/POUs/Write/MC_WriteSystemVariable/MC_WriteSystemVariableFB
/// Write specific parameter of the robot
FUNCTION_BLOCK MC_WriteSystemVariableFB EXTENDS RobotLibraryBaseExecuteFB
// ------------------------------------------------------------------------- 
//  SRCI Robot Library                                                
// ------------------------------------------------------------------------- 
//                                                                           
//  Object:      WriteSystemVariableFB                                       
//  Author:      Thorsten Brach                                                
//  Date:        2024-06-01
//
//  Description:                                              
//   
//                                                                           
//  Copyright: 
//    (C) 2024 Thorsten Brach. All rights reserved                                                                                                                                            
//             Licensed under the LGPL-3.0 license.
//                                                                           
//  Disclaimer:                                                                           
//    This project is provided without any guarantee and can be used for   
//    private and commercial purposes. Any use is at the user’s 
//    own risk and responsibility.
//
// -------------------------------------------------------------------------
VAR_INPUT
  /// Processing Mode
  ProcessingMode     : ProcessingMode;
  /// Defines the target sequence in which the command will be executed
  SequenceFlag       : SequenceFlag;
  /// command parameter 
  ParCmd             : WriteSystemVariableParCmd;
END_VAR
VAR_OUTPUT
  /// Command is transferred and confirmed by the RC
  CommandBuffered    : BOOL;
  /// The command was aborted by another command.
  CommandAborted     : BOOL;
  /// TRUE, while command is interrupted during execution and can be continued
  CommandInterrupted : BOOL;
  /// TRUE, when parameters were overwritten but not activated on RC until a restart of the RC
  RestartRequested   : BOOL;
  /// command outputs
  OutCmd             : WriteSystemVariableOutCmd;       
END_VAR

VAR
  /// internal copy of command parameter 
 _parCmd             : WriteSystemVariableParCmd;
  /// command data to send
 _command            : WriteSystemVariableSendData;
  /// response data received
 _response           : WriteSystemVariableRecvData;      
END_VAR

SUPER^(AxesGroup := AxesGroup);

METHOD PROTECTED CheckFunctionSupported : BOOL
VAR_IN_OUT
  /// Robot assignment of function
  AxesGroup : AxesGroup; 
END_VAR
CheckFunctionSupported := AxesGroup.InternalData.RCSupportedFunctions.WriteSystemVariable;

IF ( NOT CheckFunctionSupported )
THEN
  // call base implementation for set error and create log entry
  SUPER^.CheckFunctionSupported(AxesGroup := AxesGroup);
END_IF
END_METHOD

METHOD PROTECTED CheckParameterChanged : BOOL
VAR_IN_OUT
  /// Robot assignment of function
  AxesGroup    : AxesGroup; 
END_VAR
// Check ParCmd Size is > 0, because MemCmp does not work correctly with size = 0
IF (SIZEOF(ParCmd) = 0) 
THEN 
  RETURN;
END_IF

// compare memory 
_parameterChanged := ( SysDepMemCmp(pData1 := ADR(ParCmd), pData2 := ADR(_parCmd), DataLen := SIZEOF(ParCmd)) <> RobotLibraryConstants.OK );

// check parameter valid ?
_parameterValid   := CheckParameterValid( AxesGroup := AxesGroup );

IF ((  _parameterChanged        )  AND 
    (  _parameterValid          )) OR
    (  _parameterUpdateInternal )  
THEN  
  // reset internal flag for send parameter update
 _parameterUpdateInternal := FALSE;
  // update internal copy of parameters 
 _parCmd := ParCmd;
  // inc parameter sequence
 _command.ParSeq := _command.ParSeq + 1;
  // update command data  
  CommandData := CreateCommandPayload(AxesGroup := AxesGroup); // ( Access via reference to rCommandFB in ACR )
  // notify active command register 
  AxesGroup.Acyclic.ActiveCommandRegister.NotifyParameterChanged := _uniqueID;
END_IF
END_METHOD

METHOD INTERNAL CreateCommandPayload : RobotLibrarySendDataFB
VAR_IN_OUT
  /// Robot assignment of function
  AxesGroup : AxesGroup; 
END_VAR
// Table 6-626: Sent CMD payload (PLC to RC) of "WriteSystemVariable"
// --------------------------
// Header
// --------------------------
// Byte 00 : UINT  - Type HB     
// Byte 01 :       - Type LB    
// Byte 02 : USINT - Reserve | ExecutionMode
// Byte 03 : USINT - ParSeq  | Priority
// --------------------------
// Datablock
// --------------------------
// Byte 04 : SINT EmitterID[0]
// Byte 05 : SINT EmitterID[1]
// Byte 06 : SINT EmitterID[2]
// Byte 07 : SINT EmitterID[3]
// Byte 08 : SINT ListenerID
// Byte 09 : BYTE Reserved
// Byte 10 : UINT ParameterID[0]
// Byte 11 : 
// Byte 12 : UINT ParameterID[1]
// Byte 13 : 
// Byte 14 : UINT ParameterID[2]
// Byte 15 : 
// Byte 16 : UINT ParameterID[3]
// Byte 17 : 
// Byte 18 : UINT ParameterID[4]
// Byte 19 : 
// Byte 20 : UINT ParameterID[5]
// Byte 21 : 
// Byte 22 : UINT ParameterID[6]
// Byte 23 : 
// Byte 24 : UINT ParameterID[7]
// Byte 25 : 
// Byte 26 : USINT SubParameterID[0]
// Byte 27 : USINT SubParameterID[1]
// Byte 28 : USINT SubParameterID[2]
// Byte 29 : USINT SubParameterID[3]
// Byte 30 : USINT SubParameterID[4]
// Byte 31 : USINT SubParameterID[5]
// Byte 32 : USINT SubParameterID[6]
// Byte 33 : USINT SubParameterID[7]
// Byte 34 : USINT DataType[0]
// Byte 35 : USINT DataType[1]
// Byte 36 : USINT DataType[2]
// Byte 37 : USINT DataType[3]
// Byte 38 : USINT DataType[4]
// Byte 39 : USINT DataType[5]
// Byte 40 : USINT DataType[6]
// Byte 41 : USINT DataType[7]
// Byte 42 : BYTE Data_0[0]
// Byte 43 : BYTE Data_0[1]
// Byte 44 : BYTE Data_0[2]
// Byte 45 : BYTE Data_0[3]
// Byte 46 : BYTE Data_1[0]
// Byte 47 : BYTE Data_1[1]
// Byte 48 : BYTE Data_1[2]
// Byte 49 : BYTE Data_1[3]
// Byte 50 : BYTE Data_2[0]
// Byte 51 : BYTE Data_2[1]
// Byte 52 : BYTE Data_2[2]
// Byte 53 : BYTE Data_2[3]
// Byte 54 : BYTE Data_3[0]
// Byte 55 : BYTE Data_3[1]
// Byte 56 : BYTE Data_3[2]
// Byte 57 : BYTE Data_3[3]
// Byte 58 : BYTE Data_4[0]
// Byte 59 : BYTE Data_4[1]
// Byte 60 : BYTE Data_4[2]
// Byte 61 : BYTE Data_4[3]
// Byte 62 : BYTE Data_5[0]
// Byte 63 : BYTE Data_5[1]
// Byte 64 : BYTE Data_5[2]
// Byte 65 : BYTE Data_5[3]
// Byte 66 : BYTE Data_6[0]
// Byte 67 : BYTE Data_6[1]
// Byte 68 : BYTE Data_6[2]
// Byte 69 : BYTE Data_6[3]
// Byte 70 : BYTE Data_7[0]
// Byte 71 : BYTE Data_7[1]
// Byte 72 : BYTE Data_7[2]
// Byte 73 : BYTE Data_7[3]
// Byte 74 : BOOL RCParameter
// --------------------------

VAR
  /// internal index for loops
  _idx : DINT;
END_VAR
// set command parameter 
_command.CmdTyp         :=  CmdType.WriteSystemVariable;
_command.ExecMode       :=  ExecMode;
_command.ParSeq         := _command.ParSeq;
_command.Priority       :=  Priority;
                        
_command.EmitterID[0]   :=  0;
_command.EmitterID[1]   :=  0;
_command.EmitterID[2]   :=  0;
_command.EmitterID[3]   :=  0;
_command.ListenerID     :=  _parCmd.ListenerID;
_command.Reserve        :=  0;
_command.ParameterID    :=  _parCmd.ParameterID;
_command.SubParameterID :=  _parCmd.SubParameterID;
_command.DataType       :=  _parCmd.DataType;
_command.Data_0         :=  _parCmd.Data_0;
_command.Data_1         :=  _parCmd.Data_1;
_command.Data_2         :=  _parCmd.Data_2;
_command.Data_3         :=  _parCmd.Data_3;
_command.Data_4         :=  _parCmd.Data_4;
_command.Data_5         :=  _parCmd.Data_5;
_command.Data_6         :=  _parCmd.Data_6;
_command.Data_7         :=  _parCmd.Data_7;


// copy command data to header
_cmdHeader := _command;
// call base implementation to copy header to payload buffer
CreateCommandPayload := SUPER^.CreateCommandPayload(AxesGroup := AxesGroup);

// add command.EmitterID[0]
CreateCommandPayload.AddSint(_command.EmitterID[0]);
// add command.EmitterID[1]
CreateCommandPayload.AddSint(_command.EmitterID[1]);
// add command.EmitterID[2]
CreateCommandPayload.AddSint(_command.EmitterID[2]);
// add command.EmitterID[3]
CreateCommandPayload.AddSint(_command.EmitterID[3]);
// add command.ListenerID
CreateCommandPayload.AddSint(_command.ListenerID);
// add command.Reserve
CreateCommandPayload.AddByte(_command.Reserve);

FOR _idx := 0 TO 7 
DO
  // add command.ParameterID[_idx]
  CreateCommandPayload.AddUint(_command.ParameterID[_idx]);
END_FOR

FOR _idx := 0 TO 7 
DO
  // add command.SubParameterID[_idx]
  CreateCommandPayload.AddUsint(_command.SubParameterID[_idx]);
END_FOR

FOR _idx := 0 TO 7 
DO
  // add command.DataType[_idx]
  CreateCommandPayload.AddUsint(_command.DataType[_idx]);
END_FOR

FOR _idx := 0 TO 3 
DO
  // add command.Data_0[_idx]
  CreateCommandPayload.AddUsint(_command.Data_0[_idx]);
END_FOR

FOR _idx := 0 TO 3 
DO
  // add command.Data_1[_idx]
  CreateCommandPayload.AddUsint(_command.Data_1[_idx]);
END_FOR

FOR _idx := 0 TO 3 
DO
  // add command.Data_2[_idx]
  CreateCommandPayload.AddUsint(_command.Data_2[_idx]);
END_FOR

FOR _idx := 0 TO 3 
DO
  // add command.Data_3[_idx]
  CreateCommandPayload.AddUsint(_command.Data_3[_idx]);
END_FOR

FOR _idx := 0 TO 3 
DO
  // add command.Data_4[_idx]
  CreateCommandPayload.AddUsint(_command.Data_4[_idx]);
END_FOR

FOR _idx := 0 TO 3 
DO
  // add command.Data_5[_idx]
  CreateCommandPayload.AddUsint(_command.Data_5[_idx]);
END_FOR

FOR _idx := 0 TO 3 
DO
  // add command.Data_6[_idx]
  CreateCommandPayload.AddUsint(_command.Data_6[_idx]);
END_FOR

FOR _idx := 0 TO 3 
DO
  // add command.Data_7[_idx]
  CreateCommandPayload.AddUsint(_command.Data_7[_idx]);
END_FOR

// Create logging
CreateCommandPayloadLog(AxesGroup := AxesGroup);
END_METHOD

METHOD INTERNAL CreateCommandPayloadLog
VAR_IN_OUT
  /// Robot assignment of function
  AxesGroup : AxesGroup; 
END_VAR
VAR 
  /// internal index for loops
 _idx : DINT;
END_VAR
// Create log entry for Parameter start
CreateLogMessage      ( Timestamp   := AxesGroup.InternalData.SystemTime,
                        MessageType := MessageType.CMD,
                        Severity    := Severity.DEBUG,
                        MessageCode := 0,
                        MessageText := 'Create command payload with the following parameter(s) :');
  
// Create log entry for EmitterID[x]
FOR _idx := 0 TO 3
DO
  CreateLogMessagePara2 ( Timestamp   := AxesGroup.InternalData.SystemTime,
                          MessageType := MessageType.CMD,
                          Severity    := Severity.DEBUG,
                          MessageCode := 0,
                          MessageText := 'Command.EmitterID[{2}] = {1}',
                          Para1       :=  SINT_TO_STRING(_command.EmitterID[_idx]),
                          Para2       :=  DINT_TO_STRING(_idx));
END_FOR

// Create log entry for ListenerID
CreateLogMessagePara1 ( Timestamp   := AxesGroup.InternalData.SystemTime,
                        MessageType := MessageType.CMD,
                        Severity    := Severity.DEBUG,
                        MessageCode := 0,
                        MessageText := 'Command.ListenerID = {1}',
                        Para1       :=  SINT_TO_STRING(_command.ListenerID));
                        
// Create log entry for Reserve
CreateLogMessagePara1 ( Timestamp   := AxesGroup.InternalData.SystemTime,
                        MessageType := MessageType.CMD,
                        Severity    := Severity.DEBUG,
                        MessageCode := 0,
                        MessageText := 'Command.Reserve = {1}',
                        Para1       :=  BYTE_TO_STRING(_command.Reserve));
                       
                       
// Create log entry for ParameterID[_idx]
FOR _idx := 0 TO 7
DO
  CreateLogMessagePara2 ( Timestamp   := AxesGroup.InternalData.SystemTime,
                          MessageType := MessageType.CMD,
                          Severity    := Severity.DEBUG,
                          MessageCode := 0,
                          MessageText := 'Command.ParameterID[{2}] = {1}',
                          Para1       :=  UINT_TO_STRING(_command.ParameterID[_idx]),
                          Para2       :=  DINT_TO_STRING(_idx));
END_FOR

// Create log entry for SubParameterID[_idx]
FOR _idx := 0 TO 7
DO
  CreateLogMessagePara2 ( Timestamp   := AxesGroup.InternalData.SystemTime,
                          MessageType := MessageType.CMD,
                          Severity    := Severity.DEBUG,
                          MessageCode := 0,
                          MessageText := 'Command.SubParameterID[{2}] = {1}',
                          Para1       :=  USINT_TO_STRING(_command.SubParameterID[_idx]),
                          Para2       :=  DINT_TO_STRING(_idx));
END_FOR
                       
// Create log entry for DataType[_idx]
FOR _idx := 0 TO 7
DO
  CreateLogMessagePara2 ( Timestamp   := AxesGroup.InternalData.SystemTime,
                          MessageType := MessageType.CMD,
                          Severity    := Severity.DEBUG,
                          MessageCode := 0,
                          MessageText := 'Command.DataType[{2}] = {1}',
                          Para1       :=  USINT_TO_STRING(_command.DataType[_idx]),
                          Para2       :=  DINT_TO_STRING(_idx));
END_FOR

// Create log entry for Data_0[_idx]
FOR _idx := 0 TO 3
DO
  CreateLogMessagePara2 ( Timestamp   := AxesGroup.InternalData.SystemTime,
                          MessageType := MessageType.CMD,
                          Severity    := Severity.DEBUG,
                          MessageCode := 0,
                          MessageText := 'Command.Data_0[{2}] = {1}',
                          Para1       :=  BYTE_TO_STRING(_command.Data_0[_idx]),
                          Para2       :=  DINT_TO_STRING(_idx));
END_FOR

// Create log entry for Data_1[_idx]
FOR _idx := 0 TO 3
DO
  CreateLogMessagePara2 ( Timestamp   := AxesGroup.InternalData.SystemTime,
                          MessageType := MessageType.CMD,
                          Severity    := Severity.DEBUG,
                          MessageCode := 0,
                          MessageText := 'Command.Data_1[{2}] = {1}',
                          Para1       :=  BYTE_TO_STRING(_command.Data_1[_idx]),
                          Para2       :=  DINT_TO_STRING(_idx));
END_FOR

// Create log entry for Data_2[_idx]
FOR _idx := 0 TO 3
DO
  CreateLogMessagePara2 ( Timestamp   := AxesGroup.InternalData.SystemTime,
                          MessageType := MessageType.CMD,
                          Severity    := Severity.DEBUG,
                          MessageCode := 0,
                          MessageText := 'Command.Data_2[{2}] = {1}',
                          Para1       :=  BYTE_TO_STRING(_command.Data_2[_idx]),
                          Para2       :=  DINT_TO_STRING(_idx));
END_FOR

// Create log entry for Data_3[_idx]
FOR _idx := 0 TO 3
DO
  CreateLogMessagePara2 ( Timestamp   := AxesGroup.InternalData.SystemTime,
                          MessageType := MessageType.CMD,
                          Severity    := Severity.DEBUG,
                          MessageCode := 0,
                          MessageText := 'Command.Data_3[{2}] = {1}',
                          Para1       :=  BYTE_TO_STRING(_command.Data_3[_idx]),
                          Para2       :=  DINT_TO_STRING(_idx));
END_FOR

// Create log entry for Data_4[_idx]
FOR _idx := 0 TO 3
DO
  CreateLogMessagePara2 ( Timestamp   := AxesGroup.InternalData.SystemTime,
                          MessageType := MessageType.CMD,
                          Severity    := Severity.DEBUG,
                          MessageCode := 0,
                          MessageText := 'Command.Data_4[{2}] = {1}',
                          Para1       :=  BYTE_TO_STRING(_command.Data_4[_idx]),
                          Para2       :=  DINT_TO_STRING(_idx));
END_FOR

// Create log entry for Data_5[_idx]
FOR _idx := 0 TO 3
DO
  CreateLogMessagePara2 ( Timestamp   := AxesGroup.InternalData.SystemTime,
                          MessageType := MessageType.CMD,
                          Severity    := Severity.DEBUG,
                          MessageCode := 0,
                          MessageText := 'Command.Data_5[{2}] = {1}',
                          Para1       :=  BYTE_TO_STRING(_command.Data_5[_idx]),
                          Para2       :=  DINT_TO_STRING(_idx));
END_FOR

// Create log entry for Data_6[_idx]
FOR _idx := 0 TO 3
DO
  CreateLogMessagePara2 ( Timestamp   := AxesGroup.InternalData.SystemTime,
                          MessageType := MessageType.CMD,
                          Severity    := Severity.DEBUG,
                          MessageCode := 0,
                          MessageText := 'Command.Data_6[{2}] = {1}',
                          Para1       :=  BYTE_TO_STRING(_command.Data_6[_idx]),
                          Para2       :=  DINT_TO_STRING(_idx));
END_FOR

// Create log entry for Data_7[_idx]
FOR _idx := 0 TO 3
DO
  CreateLogMessagePara2 ( Timestamp   := AxesGroup.InternalData.SystemTime,
                          MessageType := MessageType.CMD,
                          Severity    := Severity.DEBUG,
                          MessageCode := 0,
                          MessageText := 'Command.Data_7[{2}] = {1}',
                          Para1       :=  BYTE_TO_STRING(_command.Data_7[_idx]),
                          Para2       :=  DINT_TO_STRING(_idx));
END_FOR
END_METHOD

METHOD FB_init : BOOL
VAR_INPUT
  /// if TRUE, the retain variables are initialized (warm start / cold start)
  bInitRetains : BOOL; 
  /// if TRUE, the instance afterwards gets moved into the copy code (online change)
  bInCopyCode  : BOOL;  
END_VAR
MyType := 'MC_WriteSystemVariableFB';

ExecMode := ExecutionMode.PARALLEL;
END_METHOD

METHOD PROTECTED OnCall
VAR_IN_OUT
  /// Robot assignment of function
  AxesGroup : AxesGroup; 
END_VAR
// call base implementation
SUPER^.OnCall(AxesGroup := AxesGroup);

CASE _stepCmd OF
  
  00:  IF ( _execute_R.Q )  
       THEN
         // Check function is supported and parameter are valid ?
         IF (( CheckFunctionSupported( AxesGroup := AxesGroup )) AND
             ( CheckParameterValid   ( AxesGroup := AxesGroup )))
         THEN      
           // set busy flag
           Busy := TRUE;
           // Reset command outputs
           SysDepMemSet(pDest := ADR(OutCmd), Value := 0, DataLen := SIZEOF(OutCmd));         
           // apply command parameter
          _parCmd := ParCmd;
           // init parameter sequence
          _command.ParSeq := 1;
           // create command data
           CommandData := CreateCommandPayload(AxesGroup := AxesGroup);
           // Add command to active command register
          _uniqueID := AxesGroup.Acyclic.ActiveCommandRegister.AddCmd( pCommandFB := ADR(THIS^ ));     
           // set timeout
           SetTimeout(PT := _timeoutCmd, rTimer := _timerCmd);
           // inc step counter
          _stepCmd := _stepCmd + 1;
         END_IF 
       END_IF
     

  01:  // Wait for responce received
       IF ( _responseReceived )
       THEN
         // reset response received flag
        _responseReceived := FALSE;

         CASE  _response.State 
         OF
           CmdMessageState.BUFFERED    : CommandBuffered    := TRUE;
           CmdMessageState.INTERRUPTED : CommandInterrupted := TRUE;
           CmdMessageState.DONE        : Done               := TRUE;
           CmdMessageState.ABORTED     : CommandAborted     := TRUE;
           CmdMessageState.ERROR       : Error              := TRUE;
         END_CASE
                
         RestartRequested := _response.RestartRequested    ;            
         // Done, Aborted or Error ?
         IF (_response.State >= CmdMessageState.DONE )
         THEN
           // Reset Busy flag
           Busy := FALSE;
           // Update results
           OutCmd.InvocationCounter := _response.InvocationCounter;
           OutCmd.OriginID          := _response.OriginID;
           OutCmd.RestartRequested  := _response.RestartRequested;
           // set timeout
           SetTimeout(PT := _timeoutCmd, rTimer := _timerCmd);
           // inc step counter
          _stepCmd := _stepCmd + 1; 
         END_IF
       END_IF


  02: IF ( NOT Execute)
      THEN
        Reset();
      END_IF     

ELSE
  // invalid step
  ErrorID := RobotLibraryEvents.ERR_INVALID_STEP;
END_CASE


// Reset FB
IF ( NOT Execute )
THEN
  Reset();
END_IF
END_METHOD

METHOD INTERNAL ParseResponsePayload : DINT
VAR_INPUT
  /// Response data
  ResponseData : RobotLibraryRecvDataFB;
  /// Timestamp
  Timestamp    : SystemTime;  
END_VAR
// Table 6-627: Received CMD payload (RC to PLC) of "WriteSystemVariable"
// --------------------------
// Header
// --------------------------
// Byte 00 : USINT   - ParSeq | State     
// Byte 01 : SINT    - AlarmMessageSeverity    
// Byte 02 : UINT    - AlarmMessageCode HB
// Byte 03 :         - AlarmMessageCode LB
// --------------------------
// Datablock
// --------------------------
// Byte 04 : USINT      - InvocationCounter
// Byte 05 : SINT       - Reserved
// Byte 06 : INT        - OriginID HW HB
// Byte 07 :            - OriginID HW LB
// Byte 08 : BOOL       - RestartRequested
// call base implementation to parse the header from payload buffer
ResponseData.PayloadPtr := SUPER^.ParseResponsePayload(ResponseData := ResponseData, Timestamp := Timestamp);

// copy parsed header to response
_response.ParSeq               := _rspHeader.ParSeq;
_response.State                := _rspHeader.State;
_response.AlarmMessageSeverity := _rspHeader.AlarmMessageSeverity;
_response.AlarmMessageCode     := _rspHeader.AlarmMessageCode;

// Get Response.InvocationCounter
_response.InvocationCounter := ResponseData.GetUsint();
// Get Response.Reserve
_response.Reserve := ResponseData.GetSint();
// Get Response.OriginID
_response.OriginID := ResponseData.GetInt();
// Get Response.RestartRequested
_response.RestartRequested := ResponseData.GetBool();

// Create logging
ParseResponsePayloadLog(ResponseData := ResponseData, Timestamp := Timestamp);
END_METHOD

METHOD INTERNAL ParseResponsePayloadLog
VAR_INPUT
  /// Response data
  ResponseData : RobotLibraryRecvDataFB;
  /// Timestamp
  Timestamp    : SystemTime;  
END_VAR
// Create log entry for Parameter start
CreateLogMessage      ( Timestamp   := Timestamp,
                        MessageType := MessageType.CMD,
                        Severity    := Severity.DEBUG,
                        MessageCode := 0,
                        MessageText := 'Parsed the following parameter(s) from response data:');

// Create log entry for InvocationCounter
CreateLogMessagePara1 ( Timestamp   := Timestamp,
                        MessageType := MessageType.CMD,
                        Severity    := Severity.DEBUG,
                        MessageCode := 0,
                        MessageText := 'Response.InvocationCounter = {1}',
                        Para1       :=  USINT_TO_STRING(_response.InvocationCounter));

// Create log entry for Reserve
CreateLogMessagePara1 ( Timestamp   := Timestamp,
                        MessageType := MessageType.CMD,
                        Severity    := Severity.DEBUG,
                        MessageCode := 0,
                        MessageText := 'Response.Reserve = {1}',
                        Para1       :=  SINT_TO_STRING(_response.Reserve));

// Create log entry for OriginID
CreateLogMessagePara1 ( Timestamp   := Timestamp,
                        MessageType := MessageType.CMD,
                        Severity    := Severity.DEBUG,
                        MessageCode := 0,
                        MessageText := 'Response.OriginID = {1}',
                        Para1       :=  INT_TO_STRING(_response.OriginID));                       

// Create log entry for RestartRequested
CreateLogMessagePara1 ( Timestamp   := Timestamp,
                        MessageType := MessageType.CMD,
                        Severity    := Severity.DEBUG,
                        MessageCode := 0,
                        MessageText := 'Response.RestartRequested = {1}',
                        Para1       :=  BOOL_TO_STRING(_response.RestartRequested));
END_METHOD

METHOD PROTECTED Reset : DINT
VAR_INPUT
END_VAR
Reset := SUPER^.Reset();

Done               := FALSE;
Busy               := FALSE;
RestartRequested   := FALSE;
CommandBuffered    := FALSE;
CommandAborted     := FALSE;
CommandInterrupted := FALSE;
END_METHOD

END_FUNCTION_BLOCK

// Library/POUs/Write/MC_WriteToolData/MC_WriteToolDataFB
/// Change configuration of selected tool number
FUNCTION_BLOCK MC_WriteToolDataFB EXTENDS RobotLibraryBaseExecuteFB
// ------------------------------------------------------------------------- 
//  SRCI Robot Library                                                
// ------------------------------------------------------------------------- 
//                                                                           
//  Object:      WriteToolDataFB                                       
//  Author:      Thorsten Brach                                                
//  Date:        2024-06-01
//
//  Description:                                              
//   
//                                                                           
//  Copyright: 
//    (C) 2024 Thorsten Brach. All rights reserved                                                                                                                                            
//             Licensed under the LGPL-3.0 license.
//                                                                           
//  Disclaimer:                                                                           
//    This project is provided without any guarantee and can be used for   
//    private and commercial purposes. Any use is at the user’s 
//    own risk and responsibility.
//
// -------------------------------------------------------------------------
VAR_INPUT
  /// Processing Mode
  ProcessingMode     : ProcessingMode;  
  /// Defines the target sequence in which the command will be executed
  SequenceFlag       : SequenceFlag;
  /// command parameter 
  ParCmd             : WriteToolDataParCmd;
END_VAR
VAR_OUTPUT
  /// Command is transferred and confirmed by the RC
  CommandBuffered    : BOOL;
  /// The command was aborted by another command
  CommandAborted     : BOOL;
  /// TRUE, while command is interrupted during execution and can be continued.
  CommandInterrupted : BOOL;
  /// command outputs
  OutCmd             : WriteToolDataOutCmd;       
END_VAR

VAR
  /// internal copy of command parameter 
 _parCmd             : WriteToolDataParCmd;
  /// command data to send
 _command            : WriteToolDataSendData;
  /// response data received
 _response           : WriteToolDataRecvData;      
END_VAR

SUPER^(AxesGroup := AxesGroup);

METHOD PROTECTED CheckFunctionSupported : BOOL
VAR_IN_OUT
  /// Robot assignment of function
  AxesGroup : AxesGroup; 
END_VAR
CheckFunctionSupported := AxesGroup.InternalData.RCSupportedFunctions.WriteToolData;

IF ( NOT CheckFunctionSupported )
THEN
  // call base implementation for set error and create log entry
  SUPER^.CheckFunctionSupported(AxesGroup := AxesGroup);
END_IF
END_METHOD

METHOD PROTECTED CheckParameterChanged : BOOL
VAR_IN_OUT
  /// Robot assignment of function
  AxesGroup    : AxesGroup; 
END_VAR
// Check ParCmd Size is > 0, because MemCmp does not work correctly with size = 0
IF (SIZEOF(ParCmd) = 0) 
THEN 
  RETURN;
END_IF

// compare memory 
_parameterChanged := ( SysDepMemCmp(pData1 := ADR(ParCmd), pData2 := ADR(_parCmd), DataLen := SIZEOF(ParCmd)) <> RobotLibraryConstants.OK );

// check parameter valid ?
_parameterValid   := CheckParameterValid( AxesGroup := AxesGroup );

IF ((  _parameterChanged        )  AND 
    (  _parameterValid          )) OR
    (  _parameterUpdateInternal )  
THEN  
  // reset internal flag for send parameter update
 _parameterUpdateInternal := FALSE;
  // update internal copy of parameters 
 _parCmd := ParCmd;
  // inc parameter sequence
 _command.ParSeq := _command.ParSeq + 1;
  // update command data  
  CommandData := CreateCommandPayload(AxesGroup := AxesGroup); // ( Access via reference to rCommandFB in ACR )
  // notify active command register 
  AxesGroup.Acyclic.ActiveCommandRegister.NotifyParameterChanged := _uniqueID;
END_IF
END_METHOD

METHOD INTERNAL CreateCommandPayload : RobotLibrarySendDataFB
VAR_IN_OUT
  /// Robot assignment of function
  AxesGroup : AxesGroup; 
END_VAR
// Table 6-126: Sent CMD payload (PLC to RC) of "WriteToolData"
// --------------------------
// Header
// --------------------------
// Byte 00 : UINT  - Type HB     
// Byte 01 :       - Type LB    
// Byte 02 : USINT - Reserve | ExecutionMode
// Byte 03 : USINT - ParSeq  | Priority
// --------------------------
// Datablock
// --------------------------
// Byte 04 : DATE ToolData.Date
// Byte 05 : 
// Byte 06 : TIME_OF_DAY ToolData.Time
// Byte 07 : 
// Byte 08 : 
// Byte 09 : REAL ToolData.X
// Byte 10 : 
// Byte 11 : 
// Byte 12 : REAL ToolData.Y
// Byte 13 : 
// Byte 14 : 
// Byte 15 : REAL ToolData.Z
// Byte 16 : 
// Byte 17 : 
// Byte 18 : REAL ToolData.RX
// Byte 19 : 
// Byte 20 : 
// Byte 21 : REAL ToolData.RY
// Byte 22 : 
// Byte 23 : 
// Byte 24 : REAL ToolData.RZ
// Byte 25 : 
// Byte 26 : 
// Byte 27 : USINT ToolData.ID
// Byte 28 : USINT ToolData.LoadNo
// Byte 29 : BOOL ToolData.ExternalTCP
// Byte 30 : BYTE Reserved
// Byte 31 : USINT ToolNo
// --------------------------
// set command parameter 
_command.CmdTyp   :=  CmdType.WriteToolData;
_command.ExecMode :=  ExecMode;
_command.ParSeq   := _command.ParSeq;
_command.Priority :=  Priority;                  
_command.ToolData :=  _parCmd.ToolData;
_command.ToolNo   :=  _parCmd.ToolNo;


// copy command data to header
_cmdHeader := _command;
// call base implementation to copy header to payload buffer
CreateCommandPayload := SUPER^.CreateCommandPayload(AxesGroup := AxesGroup);

// add command.ToolData.Timestamp.IEC_DATE
CreateCommandPayload.AddUint(_command.ToolData.Timestamp.IEC_DATE);
// add command.ToolData.Timestamp.IEC_TIME
CreateCommandPayload.AddTime(_command.ToolData.Timestamp.IEC_TIME);
// add command.ToolData.X
CreateCommandPayload.AddReal(_command.ToolData.X);
// add command.ToolData.Y
CreateCommandPayload.AddReal(_command.ToolData.Y);
// add command.ToolData.Z
CreateCommandPayload.AddReal(_command.ToolData.Z);
// add command.ToolData.Rx
CreateCommandPayload.AddReal(_command.ToolData.Rx);
// add command.ToolData.Ry
CreateCommandPayload.AddReal(_command.ToolData.Ry);
// add command.ToolData.Rz
CreateCommandPayload.AddReal(_command.ToolData.Rz);
// add command.ToolData.ID
CreateCommandPayload.AddUsint(_command.ToolData.ID);
// add command.ToolData.LoadNo
CreateCommandPayload.AddUsint(_command.ToolData.LoadNo);
// add command.ToolData.ExternalTCP
CreateCommandPayload.AddBool(_command.ToolData.ExternalTCP);
// add command.ToolData.Reserve
CreateCommandPayload.AddByte(_command.Reserve);
// add command.ToolData.ToolNo
CreateCommandPayload.AddUsint(_command.ToolNo);

// Create logging
CreateCommandPayloadLog(AxesGroup := AxesGroup);
END_METHOD

METHOD INTERNAL CreateCommandPayloadLog
VAR_IN_OUT
  /// Robot assignment of function
  AxesGroup : AxesGroup; 
END_VAR
// Create log entry for Parameter start
CreateLogMessage      ( Timestamp   := AxesGroup.InternalData.SystemTime,
                        MessageType := MessageType.CMD,
                        Severity    := Severity.DEBUG,
                        MessageCode := 0,
                        MessageText := 'Create command payload with the following parameter(s) :');
  
// Create log entry for ToolData.Timestamp.IEC_DATE
CreateLogMessagePara1 ( Timestamp   := AxesGroup.InternalData.SystemTime,
                        MessageType := MessageType.CMD,
                        Severity    := Severity.DEBUG,
                        MessageCode := 0,
                        MessageText := 'Command.ToolData.Timestamp.IEC_DATE = {1}',
                        Para1       :=  IEC_DATE_TO_STRING(_command.ToolData.Timestamp.IEC_DATE));

// Create log entry for ToolData.Timestamp.IEC_TIME
CreateLogMessagePara1 ( Timestamp   := AxesGroup.InternalData.SystemTime,
                        MessageType := MessageType.CMD,
                        Severity    := Severity.DEBUG,
                        MessageCode := 0,
                        MessageText := 'Command.ToolData.Timestamp.IEC_TIME = {1}',
                        Para1       :=  IEC_TIME_TO_STRING(_command.ToolData.Timestamp.IEC_TIME));

// Create log entry for ToolData.X
CreateLogMessagePara1 ( Timestamp   := AxesGroup.InternalData.SystemTime,
                        MessageType := MessageType.CMD,
                        Severity    := Severity.DEBUG,
                        MessageCode := 0,
                        MessageText := 'Command.ToolData.X = {1}',
                        Para1       :=  REAL_TO_STRING(_command.ToolData.X));

// Create log entry for ToolData.Y
CreateLogMessagePara1 ( Timestamp   := AxesGroup.InternalData.SystemTime,
                        MessageType := MessageType.CMD,
                        Severity    := Severity.DEBUG,
                        MessageCode := 0,
                        MessageText := 'Command.ToolData.Y = {1}',
                        Para1       :=  REAL_TO_STRING(_command.ToolData.Y));

// Create log entry for ToolData.Z
CreateLogMessagePara1 ( Timestamp   := AxesGroup.InternalData.SystemTime,
                        MessageType := MessageType.CMD,
                        Severity    := Severity.DEBUG,
                        MessageCode := 0,
                        MessageText := 'Command.ToolData.Z = {1}',
                        Para1       :=  REAL_TO_STRING(_command.ToolData.Z));

// Create log entry for ToolData.Rx
CreateLogMessagePara1 ( Timestamp   := AxesGroup.InternalData.SystemTime,
                        MessageType := MessageType.CMD,
                        Severity    := Severity.DEBUG,
                        MessageCode := 0,
                        MessageText := 'Command.ToolData.Rx = {1}',
                        Para1       :=  REAL_TO_STRING(_command.ToolData.Rx));

// Create log entry for ToolData.Ry
CreateLogMessagePara1 ( Timestamp   := AxesGroup.InternalData.SystemTime,
                        MessageType := MessageType.CMD,
                        Severity    := Severity.DEBUG,
                        MessageCode := 0,
                        MessageText := 'Command.ToolData.Ry = {1}',
                        Para1       :=  REAL_TO_STRING(_command.ToolData.Ry));

// Create log entry for ToolData.Rz
CreateLogMessagePara1 ( Timestamp   := AxesGroup.InternalData.SystemTime,
                        MessageType := MessageType.CMD,
                        Severity    := Severity.DEBUG,
                        MessageCode := 0,
                        MessageText := 'Command.ToolData.Rz = {1}',
                        Para1       :=  REAL_TO_STRING(_command.ToolData.Rz));

// Create log entry for ToolData.ID
CreateLogMessagePara1 ( Timestamp   := AxesGroup.InternalData.SystemTime,
                        MessageType := MessageType.CMD,
                        Severity    := Severity.DEBUG,
                        MessageCode := 0,
                        MessageText := 'Command.ToolData.ID = {1}',
                        Para1       :=  USINT_TO_STRING(_command.ToolData.ID));
                        
// Create log entry for ToolData.LoadNo
CreateLogMessagePara1 ( Timestamp   := AxesGroup.InternalData.SystemTime,
                        MessageType := MessageType.CMD,
                        Severity    := Severity.DEBUG,
                        MessageCode := 0,
                        MessageText := 'Command.ToolData.LoadNo = {1}',
                        Para1       :=  USINT_TO_STRING(_command.ToolData.LoadNo));                        
                        
// Create log entry for ToolData.ExternalTCP
CreateLogMessagePara1 ( Timestamp   := AxesGroup.InternalData.SystemTime,
                        MessageType := MessageType.CMD,
                        Severity    := Severity.DEBUG,
                        MessageCode := 0,
                        MessageText := 'Command.ToolData.ExternalTCP = {1}',
                        Para1       :=  BOOL_TO_STRING(_command.ToolData.ExternalTCP));                                                

// Create log entry for Reserve
CreateLogMessagePara1 ( Timestamp   := AxesGroup.InternalData.SystemTime,
                        MessageType := MessageType.CMD,
                        Severity    := Severity.DEBUG,
                        MessageCode := 0,
                        MessageText := 'Command.Reserve = {1}',
                        Para1       :=  BYTE_TO_STRING(_command.Reserve));                                                
                                                                                                
// Create log entry for ToolNo
CreateLogMessagePara1 ( Timestamp   := AxesGroup.InternalData.SystemTime,
                        MessageType := MessageType.CMD,
                        Severity    := Severity.DEBUG,
                        MessageCode := 0,
                        MessageText := 'Command.ToolNo = {1}',
                        Para1       :=  USINT_TO_STRING(_command.ToolNo));
END_METHOD

METHOD FB_init : BOOL
VAR_INPUT
  /// if TRUE, the retain variables are initialized (warm start / cold start)
  bInitRetains : BOOL; 
  /// if TRUE, the instance afterwards gets moved into the copy code (online change)
  bInCopyCode  : BOOL;  
END_VAR
MyType := 'MC_WriteToolDataFB';

ExecMode := ExecutionMode.PARALLEL;
END_METHOD

METHOD PROTECTED OnCall
VAR_IN_OUT
  /// Robot assignment of function
  AxesGroup : AxesGroup; 
END_VAR
// call base implementation
SUPER^.OnCall(AxesGroup := AxesGroup);

CASE _stepCmd OF
  
  00:  IF ( _execute_R.Q )  
       THEN
         // Check function is supported and parameter are valid ?
         IF (( CheckFunctionSupported( AxesGroup := AxesGroup )) AND
             ( CheckParameterValid   ( AxesGroup := AxesGroup )))
         THEN      
           // set busy flag
           Busy := TRUE;
           // Reset command outputs
           SysDepMemSet(pDest := ADR(OutCmd), Value := 0, DataLen := SIZEOF(OutCmd));         
           // apply command parameter
          _parCmd := ParCmd;
           // init parameter sequence
          _command.ParSeq := 1;
           // create command data
           CommandData := CreateCommandPayload(AxesGroup := AxesGroup);
           // Add command to active command register
          _uniqueID := AxesGroup.Acyclic.ActiveCommandRegister.AddCmd( pCommandFB := ADR(THIS^ ));     
           // set timeout
           SetTimeout(PT := _timeoutCmd, rTimer := _timerCmd);
           // inc step counter
          _stepCmd := _stepCmd + 1;
         END_IF 
       END_IF
     

  01:  // Wait for responce received
       IF ( _responseReceived )
       THEN
         // reset response received flag
        _responseReceived := FALSE;

         CASE  _response.State 
         OF
           CmdMessageState.BUFFERED    : CommandBuffered    := TRUE;
           CmdMessageState.INTERRUPTED : CommandInterrupted := TRUE;
           CmdMessageState.DONE        : Done               := TRUE;
           CmdMessageState.ABORTED     : CommandAborted     := TRUE;
           CmdMessageState.ERROR       : Error              := TRUE;
         END_CASE
                
         // Done, Aborted or Error ?
         IF (_response.State >= CmdMessageState.DONE )
         THEN
           // Reset Busy flag
           Busy := FALSE;
           // set timeout
           SetTimeout(PT := _timeoutCmd, rTimer := _timerCmd);
           // inc step counter
          _stepCmd := _stepCmd + 1; 
         END_IF
       END_IF


  02: IF ( NOT Execute)
      THEN
        Reset(); 
      END_IF     

ELSE
  // invalid step
  ErrorID := RobotLibraryEvents.ERR_INVALID_STEP;
END_CASE


// Reset FB
IF ( NOT Execute )
THEN
  Reset(); 
END_IF
END_METHOD

METHOD INTERNAL ParseResponsePayload : DINT
VAR_INPUT
  /// Response data
  ResponseData : RobotLibraryRecvDataFB;
  /// Timestamp
  Timestamp    : SystemTime;  
END_VAR
// Table 6-127: Received CMD payload (RC to PLC) of "WriteToolData"
// --------------------------
// Header
// --------------------------
// Byte 00 : USINT   - ParSeq | State     
// Byte 01 : SINT    - AlarmMessageSeverity    
// Byte 02 : UINT    - AlarmMessageCode HB
// Byte 03 :         - AlarmMessageCode LB
// --------------------------
// Datablock
// --------------------------
// call base implementation to parse the header from payload buffer
ResponseData.PayloadPtr := SUPER^.ParseResponsePayload(ResponseData := ResponseData, Timestamp := Timestamp);

// copy parsed header to response
_response.ParSeq               := _rspHeader.ParSeq;
_response.State                := _rspHeader.State;
_response.AlarmMessageSeverity := _rspHeader.AlarmMessageSeverity;
_response.AlarmMessageCode     := _rspHeader.AlarmMessageCode;

// Create logging
ParseResponsePayloadLog(ResponseData := ResponseData, Timestamp := Timestamp);
END_METHOD

METHOD INTERNAL ParseResponsePayloadLog
VAR_INPUT
  /// Response data
  ResponseData : RobotLibraryRecvDataFB;
  /// Timestamp
  Timestamp    : SystemTime;  
END_VAR
// Create log entry for Parameter start
CreateLogMessage      ( Timestamp   := Timestamp,
                        MessageType := MessageType.CMD,
                        Severity    := Severity.DEBUG,
                        MessageCode := 0,
                        MessageText := 'Parsed the following parameter(s) from response data:');
                        
// Create log entry for no parameter 
CreateLogMessage      ( Timestamp   := Timestamp,
                        MessageType := MessageType.CMD,
                        Severity    := Severity.DEBUG,
                        MessageCode := 0,
                        MessageText := 'This command has no parameter to parse...');
END_METHOD

METHOD PROTECTED Reset : DINT
VAR_INPUT
END_VAR
Reset := SUPER^.Reset();

Done               := FALSE;
Busy               := FALSE;
CommandBuffered    := FALSE;
CommandAborted     := FALSE;
CommandInterrupted := FALSE;
END_METHOD

END_FUNCTION_BLOCK
